				CASE nRail OF
					1: GVL_Alarms.R1_Stepper_Motion_Failed.sMessage := CONCAT('Stepper rail 1 motion failed: ', sErrorMsg);
					2: GVL_Alarms.R2_Stepper_Motion_Failed.sMessage := CONCAT('Stepper rail 2 motion failed: ', sErrorMsg);
					3: GVL_Alarms.R3_Stepper_Motion_Failed.sMessage := CONCAT('Stepper rail 3 motion failed: ', sErrorMsg);
					4: GVL_Alarms.R4_Stepper_Motion_Failed.sMessage := CONCAT('Stepper rail 4 motion failed: ', sErrorMsg);
				END_CASE
			END_IF
			
			fbMoveAbs(Axis := pAxis^, Execute := FALSE);
			MoveToPosition := -1;
		END_IF
		
		IF fbMoveAbs.CommandAborted THEN
			eState := LAS_Stepper_Error;
			
			pAlarmCondition := F_GetStepperAlarmCondition(nRail, 'Motion_Interrupted');
			IF pAlarmCondition <> 0 THEN
				pAlarmCondition^ := TRUE;
				
				sErrorMsg := F_GetMC2ErrorDescription(fbMoveAbs.ErrorID);
				
				CASE nRail OF
					1: GVL_Alarms.R1_Stepper_Motion_Interrupted.sMessage := CONCAT('Stepper rail 1 motion interrupted: ', sErrorMsg);
					2: GVL_Alarms.R2_Stepper_Motion_Interrupted.sMessage := CONCAT('Stepper rail 2 motion interrupted: ', sErrorMsg);
					3: GVL_Alarms.R3_Stepper_Motion_Interrupted.sMessage := CONCAT('Stepper rail 3 motion interrupted: ', sErrorMsg);
					4: GVL_Alarms.R4_Stepper_Motion_Interrupted.sMessage := CONCAT('Stepper rail 4 motion interrupted: ', sErrorMsg);
				END_CASE
			END_IF
				
			fbMoveAbs(Axis := pAxis^, Execute := FALSE);
			MoveToPosition := -1;
			
		ELSIF fbMoveAbs.Done THEN
			eState := LAS_Stepper_Ready;
			fbMoveAbs(Axis := pAxis^, Execute := FALSE);
			MoveToPosition := 1; 
			nErrID := 0;
		END_IF
	
	LAS_Stepper_Error:
		MoveToPosition := -1; 
		
END_CASE
END_METHOD

METHOD PowerDown : BOOL
VAR
	pAlarmCondition : POINTER TO BOOL;
END_VAR
fbPower(Axis := pAxis^, Enable := FALSE);
bIsUp := FALSE;

IF (eState <> LAS_Stepper_Error) AND (eState <> LAS_Stepper_PowerError) THEN
	eState := LAS_Stepper_Idle;
END_IF
END_METHOD

METHOD Reset : INT
VAR_INPUT
    bExecute : BOOL;
END_VAR

VAR
	i : UINT;
	pAlarmCondition : POINTER TO BOOL;
	nResult : INT;
	nMoveResult : INT;
	sErrorMsg : STRING(255);
END_VAR
Reset := 0;

CASE eState OF
	LAS_Stepper_Error, LAS_Stepper_PowerError, LAS_Stepper_Ready:
		fbReset(Axis := pAxis^, Execute := bExecute);
		
		IF fbReset.Busy THEN 
			IF fbReset.Error THEN
				eState := LAS_Stepper_Error;
				nErrID := fbReset.ErrorID;
				
				pAlarmCondition := F_GetStepperAlarmCondition(nRail, 'Reset_Failed');
				IF pAlarmCondition <> 0 THEN
					pAlarmCondition^ := TRUE;
					
					sErrorMsg := F_GetMC2ErrorDescription(fbReset.ErrorID);
					
					CASE nRail OF
						1: GVL_Alarms.R1_Stepper_Reset_Failed.sMessage := CONCAT('Stepper rail 1 reset failed: ', sErrorMsg);
						2: GVL_Alarms.R2_Stepper_Reset_Failed.sMessage := CONCAT('Stepper rail 2 reset failed: ', sErrorMsg);
						3: GVL_Alarms.R3_Stepper_Reset_Failed.sMessage := CONCAT('Stepper rail 3 reset failed: ', sErrorMsg);
						4: GVL_Alarms.R4_Stepper_Reset_Failed.sMessage := CONCAT('Stepper rail 4 reset failed: ', sErrorMsg);
					END_CASE
				END_IF
				
				Reset := -1;
			END_IF
		
		ELSIF fbReset.Done THEN		
			fbReset(Axis := pAxis^, Execute := FALSE);
			
			bHoldKeepAlive := FALSE;
			
			eState := LAS_Stepper_Ready;
				
			// Clear all alarm conditions related to motion
			pAlarmCondition := F_GetStepperAlarmCondition(nRail, 'Motion_Failed');
			IF pAlarmCondition <> 0 THEN pAlarmCondition^ := FALSE; END_IF
			
			pAlarmCondition := F_GetStepperAlarmCondition(nRail, 'Homing_Failed');
			IF pAlarmCondition <> 0 THEN pAlarmCondition^ := FALSE; END_IF
			
			pAlarmCondition := F_GetStepperAlarmCondition(nRail, 'Motion_Interrupted');
			IF pAlarmCondition <> 0 THEN pAlarmCondition^ := FALSE; END_IF
			
			pAlarmCondition := F_GetStepperAlarmCondition(nRail, 'Reset_Failed');
			IF pAlarmCondition <> 0 THEN pAlarmCondition^ := FALSE; END_IF
			
			pAlarmCondition := F_GetStepperAlarmCondition(nRail, 'Stop_Failed');
			IF pAlarmCondition <> 0 THEN pAlarmCondition^ := FALSE; END_IF
			
			pAlarmCondition := F_GetStepperAlarmCondition(nRail, 'UnableToReadPosition');
			IF pAlarmCondition <> 0 THEN pAlarmCondition^ := FALSE; END_IF
			
			CASE nRail OF
				1: GVL_Alarms.R1_Stepper_Reset_Failed.sMessage := '';
				2: GVL_Alarms.R2_Stepper_Reset_Failed.sMessage := '';
				3: GVL_Alarms.R3_Stepper_Reset_Failed.sMessage := '';
				4: GVL_Alarms.R4_Stepper_Reset_Failed.sMessage := '';
			END_CASE
			
			Reset := 1;
			
		END_IF
END_CASE
END_METHOD

METHOD Stop : INT
VAR
	pAlarmCondition : POINTER TO BOOL;
	sErrorMsg : STRING(255);
END_VAR
Stop := 0;

CASE eState OF
    LAS_Stepper_Ready:
        // Already stopped
        Stop := 1;
        
    LAS_Stepper_Moving:
        fbStop(Axis := pAxis^, Execute := TRUE);
              
		IF fbStop.Error THEN
			fbStop(Axis := pAxis^, Execute := FALSE);
			eState := LAS_Stepper_Error;
			nErrID := fbStop.ErrorID;
			
			pAlarmCondition := F_GetStepperAlarmCondition(nRail, 'Stop_Failed');
			IF pAlarmCondition <> 0 THEN
				pAlarmCondition^ := TRUE;
				
				
				sErrorMsg := F_GetMC2ErrorDescription(fbStop.ErrorID);
				
				
				CASE nRail OF
					1: GVL_Alarms.R1_Stepper_Stop_Failed.sMessage := CONCAT('Stepper rail 1 stop failed: ', sErrorMsg);
					2: GVL_Alarms.R2_Stepper_Stop_Failed.sMessage := CONCAT('Stepper rail 2 stop failed: ', sErrorMsg);
					3: GVL_Alarms.R3_Stepper_Stop_Failed.sMessage := CONCAT('Stepper rail 3 stop failed: ', sErrorMsg);
					4: GVL_Alarms.R4_Stepper_Stop_Failed.sMessage := CONCAT('Stepper rail 4 stop failed: ', sErrorMsg);
				END_CASE
			END_IF
			
			Stop := -1;
            
        ELSIF fbStop.Done THEN
			fbStop(Axis := pAxis^, Execute := FALSE);
			fbMoveAbs(Axis := pAxis^, Execute := FALSE);
			eState := LAS_Stepper_Idle;
            Stop := 1; 
		END_IF
    
    LAS_Stepper_Homing :
	   fbStop(Axis := pAxis^, Execute := TRUE);
	   
	   IF fbStop.Done THEN
		   fbStop(Axis := pAxis^, Execute := FALSE);
		   fbHome(Axis := pAxis^, Execute := FALSE);
		   eState := LAS_Stepper_Idle;
		   Stop   := 1;          

	   ELSIF fbStop.Error THEN
			eState := LAS_Stepper_Error;
			nErrID := fbStop.ErrorID;
			
			pAlarmCondition := F_GetStepperAlarmCondition(nRail, 'Stop_Failed');
			IF pAlarmCondition <> 0 THEN
				pAlarmCondition^ := TRUE;
				
				sErrorMsg := F_GetMC2ErrorDescription(fbStop.ErrorID);
							
				CASE nRail OF
					1: GVL_Alarms.R1_Stepper_Stop_Failed.sMessage := CONCAT('Stepper rail 1 stop failed: ', sErrorMsg);
					2: GVL_Alarms.R2_Stepper_Stop_Failed.sMessage := CONCAT('Stepper rail 2 stop failed: ', sErrorMsg);
					3: GVL_Alarms.R3_Stepper_Stop_Failed.sMessage := CONCAT('Stepper rail 3 stop failed: ', sErrorMsg);
					4: GVL_Alarms.R4_Stepper_Stop_Failed.sMessage := CONCAT('Stepper rail 4 stop failed: ', sErrorMsg);
				END_CASE
			END_IF
			
			Stop := -1;
	   END_IF
END_CASE
END_METHOD

END_FUNCTION_BLOCK

// ---- POUs/Helper/F_GetStepperAlarmCondition.TcPOU
FUNCTION F_GetStepperAlarmCondition : POINTER TO BOOL
VAR_INPUT
    nRail : SINT;            
    sAlarmType : STRING(50);   
END_VAR
VAR
    pResult : POINTER TO BOOL;
END_VAR

//Validation
IF nRail < 1 OR nRail > 4 THEN
    F_GetStepperAlarmCondition := 0;
    RETURN;
END_IF

// Map Alarm to condition boolean
IF nRail = 1 THEN
    IF sAlarmType = 'Motion_Failed' THEN
        pResult := ADR(GVL_Alarms.R1_Stepper_Motion_Failed.bCondition);
    ELSIF sAlarmType = 'Homing_Failed' THEN
        pResult := ADR(GVL_Alarms.R1_Stepper_Homing_Failed.bCondition);
    ELSIF sAlarmType = 'Motion_Interrupted' THEN
        pResult := ADR(GVL_Alarms.R1_Stepper_Motion_Interrupted.bCondition);
    ELSIF sAlarmType = 'PowerUp_Failed' THEN
        pResult := ADR(GVL_Alarms.R1_Stepper_PowerUp_Failed.bCondition);
    ELSIF sAlarmType = 'Reset_Failed' THEN
        pResult := ADR(GVL_Alarms.R1_Stepper_Reset_Failed.bCondition);
	ELSIF sAlarmType = 'Stop_Failed' THEN
        pResult := ADR(GVL_Alarms.R1_Stepper_Stop_Failed.bCondition);
	ELSIF sAlarmType = 'UnableToReadPosition' THEN
        pResult := ADR(GVL_Alarms.R1_Stepper_UnableToReadPosition.bCondition);
    END_IF
    
ELSIF nRail = 2 THEN
    IF sAlarmType = 'Motion_Failed' THEN
        pResult := ADR(GVL_Alarms.R2_Stepper_Motion_Failed.bCondition);
    ELSIF sAlarmType = 'Homing_Failed' THEN
        pResult := ADR(GVL_Alarms.R2_Stepper_Homing_Failed.bCondition);
    ELSIF sAlarmType = 'Motion_Interrupted' THEN
        pResult := ADR(GVL_Alarms.R2_Stepper_Motion_Interrupted.bCondition);
    ELSIF sAlarmType = 'PowerUp_Failed' THEN
        pResult := ADR(GVL_Alarms.R2_Stepper_PowerUp_Failed.bCondition);
    ELSIF sAlarmType = 'Reset_Failed' THEN
        pResult := ADR(GVL_Alarms.R2_Stepper_Reset_Failed.bCondition);
	ELSIF sAlarmType = 'Stop_Failed' THEN
        pResult := ADR(GVL_Alarms.R2_Stepper_Stop_Failed.bCondition);
	ELSIF sAlarmType = 'UnableToReadPosition' THEN
        pResult := ADR(GVL_Alarms.R2_Stepper_UnableToReadPosition.bCondition);
    END_IF
    
ELSIF nRail = 3 THEN
    IF sAlarmType = 'Motion_Failed' THEN
        pResult := ADR(GVL_Alarms.R3_Stepper_Motion_Failed.bCondition);
    ELSIF sAlarmType = 'Homing_Failed' THEN
        pResult := ADR(GVL_Alarms.R3_Stepper_Homing_Failed.bCondition);
    ELSIF sAlarmType = 'Motion_Interrupted' THEN
        pResult := ADR(GVL_Alarms.R3_Stepper_Motion_Interrupted.bCondition);
    ELSIF sAlarmType = 'PowerUp_Failed' THEN
        pResult := ADR(GVL_Alarms.R3_Stepper_PowerUp_Failed.bCondition);
    ELSIF sAlarmType = 'Reset_Failed' THEN
        pResult := ADR(GVL_Alarms.R3_Stepper_Reset_Failed.bCondition);
	ELSIF sAlarmType = 'Stop_Failed' THEN
        pResult := ADR(GVL_Alarms.R3_Stepper_Stop_Failed.bCondition);
	ELSIF sAlarmType = 'UnableToReadPosition' THEN
        pResult := ADR(GVL_Alarms.R3_Stepper_UnableToReadPosition.bCondition);
    END_IF
    
ELSIF nRail = 4 THEN
    IF sAlarmType = 'Motion_Failed' THEN
        pResult := ADR(GVL_Alarms.R4_Stepper_Motion_Failed.bCondition);
    ELSIF sAlarmType = 'Homing_Failed' THEN
        pResult := ADR(GVL_Alarms.R4_Stepper_Homing_Failed.bCondition);
    ELSIF sAlarmType = 'Motion_Interrupted' THEN
        pResult := ADR(GVL_Alarms.R4_Stepper_Motion_Interrupted.bCondition);
    ELSIF sAlarmType = 'PowerUp_Failed' THEN
        pResult := ADR(GVL_Alarms.R4_Stepper_PowerUp_Failed.bCondition);
    ELSIF sAlarmType = 'Reset_Failed' THEN
        pResult := ADR(GVL_Alarms.R4_Stepper_Reset_Failed.bCondition);
	ELSIF sAlarmType = 'Stop_Failed' THEN
        pResult := ADR(GVL_Alarms.R4_Stepper_Stop_Failed.bCondition);
	ELSIF sAlarmType = 'UnableToReadPosition' THEN
        pResult := ADR(GVL_Alarms.R4_Stepper_UnableToReadPosition.bCondition);
    END_IF
END_IF

F_GetStepperAlarmCondition := pResult;

END_FUNCTION

// ---- POUs/Helper/F_GetMC2ErrorDescription.TcPOU
FUNCTION F_GetMC2ErrorDescription : STRING
VAR_INPUT
    nErrorID : UDINT;  
END_VAR
VAR
    sHexCode : STRING(10);
END_VAR

CASE nErrorID OF
    // ========================================
    // NO ERROR
    // ========================================
    0:
        F_GetMC2ErrorDescription := 'No error';


    // ========================================
    // GENERAL / GROUP / AXIS READY / PARAMS
    // ========================================
    16#4052:  // 16466
        F_GetMC2ErrorDescription := 'Axis not ready to operate (configuration/startup incomplete)';

    16#4200:  // 16896
        F_GetMC2ErrorDescription := 'Group ID not allowed';

    16#4220:  // 16928
        F_GetMC2ErrorDescription := 'Group/axis busy: not ready for new task';

    16#4221:  // 16929
        F_GetMC2ErrorDescription := 'Requested target velocity is not allowed';

    16#4222:  // 16930
        F_GetMC2ErrorDescription := 'Requested target position violates software limits';

    16#4223:  // 16931
        F_GetMC2ErrorDescription := 'Axis enable (controller/feed) missing';

    16#4224:  // 16932
        F_GetMC2ErrorDescription := 'Travel path smaller than one encoder increment';

    16#4225:  // 16933
        F_GetMC2ErrorDescription := 'Drive hardware not ready at start (enable/error/startup)';

    16#4226:  // 16934
        F_GetMC2ErrorDescription := 'Invalid E-Stop parameters';

    16#4227:  // 16935
        F_GetMC2ErrorDescription := 'Setpoint generator not active';

    16#4231:  // 16945
        F_GetMC2ErrorDescription := 'Target velocity <= 0.0 not allowed';

    16#4238:  // 16952
        F_GetMC2ErrorDescription := 'Velocity override outside 0–100%';

    16#4250:  // 16976
        F_GetMC2ErrorDescription := 'Axis start / position / end position type not allowed';

    16#4253:  // 16979
        F_GetMC2ErrorDescription := 'PLC reference cam released too early during homing';

    16#4254:  // 16980
        F_GetMC2ErrorDescription := 'Distance between latch and zero pulse invalid';

    16#4260:  // 16992
        F_GetMC2ErrorDescription := 'Controller enable missing at start or during motion';


    // ========================================
    // AXIS ENABLE / FEED ENABLE / TARGET LIMITS
    // ========================================
    16#4356:  // 17238
        F_GetMC2ErrorDescription := 'Controller enable not available for this axis';

    16#4357:  // 17239
        F_GetMC2ErrorDescription := 'Negative feed enable not available';

    16#4358:  // 17240
        F_GetMC2ErrorDescription := 'Positive feed enable not available';

    16#4359:  // 17241
        F_GetMC2ErrorDescription := 'Target velocity not allowed (0 or > limits)';


    // ========================================
    // SOFTWARE LIMITS / POSITION WINDOW / ENCODER QUALITY
    // ========================================
    16#4460, 16#4462:  // 17504, 17506
        F_GetMC2ErrorDescription := 'Minimum software position limit reached/violated';

    16#4461, 16#4463:  // 17505, 17507
        F_GetMC2ErrorDescription := 'Maximum software position limit reached/violated';

    16#4464:  // 17508
        F_GetMC2ErrorDescription := 'Encoder hardware error (drive/encoder reports fault)';

    16#4465:  // 17509
        F_GetMC2ErrorDescription := 'Position initialization error at startup';

    16#4466:  // 17510
        F_GetMC2ErrorDescription := 'Invalid encoder I/O data for multiple cycles';

    16#4467:  // 17511
        F_GetMC2ErrorDescription := 'Invalid actual position';


    // ========================================
    // MOTION PARAMETER ERRORS (sanity of FB inputs)
    // ========================================
    16#44C1:  // 17601
        F_GetMC2ErrorDescription := 'Invalid velocity value';

    16#44C2:  // 17602
        F_GetMC2ErrorDescription := 'Invalid acceleration value';

    16#44C3:  // 17603
        F_GetMC2ErrorDescription := 'Invalid deceleration value';

    16#44C4:  // 17604
        F_GetMC2ErrorDescription := 'Invalid jerk value';

    16#44C5:  // 17605
        F_GetMC2ErrorDescription := 'Invalid position value';


    // ========================================
    // NC-PLC / HOMING / FUNCTION BLOCK RELATED (0x4B..)
    // ========================================
    16#4B00:  // 19200
        F_GetMC2ErrorDescription := 'Axis was stopped during motion';

    16#4B01:  // 19201
        F_GetMC2ErrorDescription := 'Axis cannot be started (error, busy, protected, not ready)';

    16#4B02:  // 19202
        F_GetMC2ErrorDescription := 'Control mode not permitted';

    16#4B03:  // 19203
        F_GetMC2ErrorDescription := 'Axis is not moving (restart only valid in motion)';

    16#4B04:  // 19204
        F_GetMC2ErrorDescription := 'Mode invalid for requested command';

    16#4B05:  // 19205
        F_GetMC2ErrorDescription := 'Command not permitted';

    16#4B06:  // 19206
        F_GetMC2ErrorDescription := 'Parameter not correct (override, gear ratio, etc.)';

    16#4B07:  // 19207
        F_GetMC2ErrorDescription := 'Timeout waiting for NC feedback (axis FB timeout)';

    16#4B08:  // 19208
        F_GetMC2ErrorDescription := 'Axis in protected/coupled mode and cannot be moved';

    16#4B09:  // 19209
        F_GetMC2ErrorDescription := 'Axis is not ready and cannot be moved';

    16#4B0A:  // 19210
        F_GetMC2ErrorDescription := 'Referencing (homing) could not be started or failed';

    16#4B0B:  // 19211
        F_GetMC2ErrorDescription := 'TouchProbe trigger definition invalid';

    16#4B0C:  // 19212
        F_GetMC2ErrorDescription := 'TouchProbe: position latch was disabled';

    16#4B0D:  // 19213
        F_GetMC2ErrorDescription := 'NC state feedback timeout (no status update)';


    // ========================================
    // DRIVE ERRORS (0x455x)
    // ========================================
    16#4550:  // 17744
        F_GetMC2ErrorDescription := 'Drive error - check drive status/diagnostics';

    16#4551:  // 17745
        F_GetMC2ErrorDescription := 'Drive in error state';

    16#4552:  // 17746
        F_GetMC2ErrorDescription := 'Drive not ready to enable';


    // ========================================
    // FUNCTION BLOCK / CYCLIC CALL ISSUES
    // ========================================
    16#4600:  // 17920
        F_GetMC2ErrorDescription := 'Invalid BufferMode for this function block';

    16#4650:  // 18000
        F_GetMC2ErrorDescription := 'Function block not called cyclically';

    16#4B66:  // 19302
        F_GetMC2ErrorDescription := 'FB not called cyclically - command not monitored';


    // ========================================
    // ENCODER ERRORS (0x4800)
    // ========================================
    16#4800:  // 18432
        F_GetMC2ErrorDescription := 'Encoder error';

    16#4801:  // 18433
        F_GetMC2ErrorDescription := 'Encoder hardware error';

    16#4802:  // 18434
        F_GetMC2ErrorDescription := 'Encoder initialization error';


    // ========================================
    // CONTROLLER ERRORS (0x4900)
    // ========================================
    16#4900:  // 18688
        F_GetMC2ErrorDescription := 'Controller error';

    16#4901:  // 18689
        F_GetMC2ErrorDescription := 'Controller not initialized';


    // ========================================
    // COUPLING / CAM / TABLE (only common ones)
    // ========================================
    16#4A01:  // 18945
        F_GetMC2ErrorDescription := 'Master axis in error during coupled motion';

    16#4A02:  // 18946
        F_GetMC2ErrorDescription := 'Slave axis in error during coupled motion';

    16#4A10:  // 19088
        F_GetMC2ErrorDescription := 'Cam plate / motion table invalid';


    // ========================================
    // FALLBACK FOR UNKNOWN CODES
    // ========================================
    ELSE
        sHexCode := DWORD_TO_HEXSTR(nErrorID, 4, FALSE);
        F_GetMC2ErrorDescription := CONCAT('MC2 Error 0x', sHexCode);
        F_GetMC2ErrorDescription := CONCAT(F_GetMC2ErrorDescription, ' (');
        F_GetMC2ErrorDescription := CONCAT(F_GetMC2ErrorDescription, UDINT_TO_STRING(nErrorID));
        F_GetMC2ErrorDescription := CONCAT(F_GetMC2ErrorDescription, ') - Check Beckhoff NC Error Codes manual');
END_CASE

END_FUNCTION

// ---- POUs/Helper/F_ValidateCommand.TcPOU
FUNCTION F_ValidateCommand : BOOL
VAR_INPUT
    sInput : STRING;
END_VAR
VAR_OUTPUT
    bIsValid : BOOL;
    nX : SINT;
    sY : STRING;
	sZ : STRING;
END_VAR
VAR
    nFirstUnderscorePos : INT;
	nSecondUnderScorePos: INT;
    sNumber : STRING;
	sRemainder : STRING;
END_VAR

bIsValid := FALSE;
nX := 0;
sY := '';
sZ := '';

// Check if string starts with "R"
IF LEFT(sInput, 1) <> 'R' THEN
    RETURN;
END_IF;

// Find the underscore position
nFirstUnderscorePos := FIND(sInput, '_');
IF nFirstUnderscorePos = 0 THEN
    RETURN;
END_IF;

// Extract the digit (X) between "R" and "_"
sNumber := MID(sInput, 1, nFirstUnderscorePos - 1);
nX := STRING_TO_SINT(sNumber);
IF nX < 1 OR nX > 4 THEN
    RETURN;
END_IF;

sRemainder := RIGHT(sInput, LEN(sInput) - nFirstUnderscorePos);
nSecondUnderscorePos := FIND(sRemainder, '_');

// Extract Y 
IF nSecondUnderscorePos = 0 THEN
    sY := RIGHT(sInput, LEN(sInput) - nFirstUnderscorePos);
ELSE
    sY := LEFT(sRemainder, nSecondUnderscorePos - 1);
    
    sZ := RIGHT(sRemainder, LEN(sRemainder) - nSecondUnderscorePos);
    
    // Check Z validity 
    IF sZ <> 'Reset' THEN
        sZ := '';  
        RETURN;    
    END_IF;
END_IF;

// Check if Y is one of the allowed values
IF sY = 'Chariot' OR 
   sY = 'Compressor' OR 
   sY = 'Sensor' OR 
   sY = 'HeatExCoupola' OR 
   sY = 'RegenCoupola' OR
   sY = 'Home' OR 
   sY = 'SetHome' OR
   sY = 'Motor' THEN
    bIsValid := TRUE;
ELSE
    sY := '';  
    sZ := '';  
END_IF;

F_ValidateCommand := bIsValid;

END_FUNCTION

// ---- POUs/Helper/F_GetLinearCommandValue.TcPOU
FUNCTION F_GetLinearCommandValue : POINTER TO FB_LinearActuator
VAR_INPUT
    nX : SINT;
    sY : STRING;
END_VAR
VAR
    i : INT;
    pResult: POINTER TO FB_LinearActuator;
END_VAR

FOR i := 1 TO nEntryCount DO
    IF aLookupTable[i].nX = nX AND aLookupTable[i].sY = sY THEN
			pResult := aLookupTable[i].sValue;
        EXIT;
    END_IF;
END_FOR;

F_GetLinearCommandValue := pResult;

END_FUNCTION

// ---- POUs/Helper/F_GetLinearCommandMember.TcPOU
FUNCTION F_GetLinearCommandmember : POINTER TO ST_LinearActuatorCommand
VAR_INPUT
    nX : SINT;
    sY : STRING;
END_VAR
VAR
    i : INT;
    pResult: POINTER TO ST_LinearActuatorCommand;
END_VAR

FOR i := 1 TO nEntryCount DO
    IF aLookupTable[i].nX = nX AND aLookupTable[i].sY = sY THEN
			pResult := aLookupTable[i].sCommand;
        EXIT;
    END_IF;
END_FOR;

F_GetLinearCommandMember := pResult;

END_FUNCTION

// ---- POUs/Helper/F_GetStepperCommandValue.TcPOU
FUNCTION F_GetStepperCommandValue : POINTER TO FB_StepperMotor
VAR_INPUT
    nX : SINT;
    sY : STRING;
END_VAR
VAR
    i : INT;
    pResult: POINTER TO FB_StepperMotor;
END_VAR

FOR i := 1 TO nEntryCount DO
    IF aLookupTable[i].nX = nX AND aLookupTable[i].sY = sY THEN
			pResult := aLookupTable[i].sValue;
        EXIT;
    END_IF;
END_FOR;

F_GetStepperCommandValue := pResult;

END_FUNCTION

// ---- POUs/Helper/F_GetStepperCommandMember.TcPOU
FUNCTION F_GetStepperCommandMember : POINTER TO ST_StepperMotorCommand
VAR_INPUT
    nX : SINT;
    sY : STRING;
END_VAR
VAR
    i : INT;
    pResult: POINTER TO ST_StepperMotorCommand;
END_VAR

FOR i := 1 TO nEntryCount DO
    IF aLookupTable[i].nX = nX AND aLookupTable[i].sY = sY THEN
			pResult := aLookupTable[i].sCommand;
        EXIT;
    END_IF;
END_FOR;

F_GetStepperCommandMember := pResult;

END_FUNCTION
